FUNCTION_BLOCK PUBLIC Cylinder
VAR_INPUT
END_VAR
VAR_OUTPUT
END_VAR
VAR
END_VAR

END_FUNCTION_BLOCK

(* stored: Version 1.1.0.1, ProductVersion 3.1.4024.16
   POU Cylinder: Id {f6a3a8d9-e4ba-4cdf-b01a-dbe0b512db31}, SpecialFunc None *)
